// TIA Portal V18 export
FUNCTION_BLOCK "P01_TCP_Com"   // FB12, LAD
{ S7_Optimized_Access := 'FALSE' }
// stored: SetENOAutomatically false
   VAR_INPUT
      I_Modbus_Slave_Addr : Byte;
      I_Start : Bool;
      I_Frequency : Real;   // 0-100（%）
   END_VAR
   VAR
      FB_Always_True : Bool;
      Start_TSEND_C { S7_SetPoint := 'True'} : TSEND_C;
      Frequency_TSNED_C { S7_SetPoint := 'True'} : TSEND_C;
      P1 : Bool;
      P2 : Bool;
      Start_T { S7_SetPoint := 'True'} : TON_TIME;
      Stop_T { S7_SetPoint := 'True'} : TOF_TIME;
      Command_Start { S7_SetPoint := 'True'} : Bool;
      Command_Stop { S7_SetPoint := 'True'} : Bool;
      Command_Freq { S7_SetPoint := 'True'} : Bool;
      Start_Array : Array[0..5] of Byte;
      Stop_Array : Array[0..5] of Byte;
      Freq_Array : Array[0..8] of Byte;
      CRC_Result : Word;
      "TSEND_DATA_Start/Stop" : Array[0..7] of Byte;
      TSEND_DATA_Freq : Array[0..10] of Byte;
      Start_TSEND_Rescan_T { S7_SetPoint := 'True'} : TON_TIME;
      Frequency_TSEND_Rescan_T { S7_SetPoint := 'True'} : TON_TIME;
      LGF_Impulse_Instance { S7_SetPoint := 'True'} : "LGF_Impulse";
   END_VAR
   VAR_TEMP
      T_Start_TSEND : Bool;
      T_Stop_TSEND : Bool;
      T_Frequency_TSEND : Bool;
      T_Frequency : Word;
   END_VAR
   // Start_Array[0] := 16#01;
   // Start_Array[1] := 16#05;
   // Start_Array[2] := 16#00;
   // Start_Array[3] := 16#04;
   // Start_Array[4] := 16#FF;
   // Start_Array[5] := 16#00;
   // Stop_Array[0] := 16#01;
   // Stop_Array[1] := 16#05;
   // Stop_Array[2] := 16#00;
   // Stop_Array[3] := 16#04;
   // Stop_Array[4..5] := 16#00;
   // Freq_Array[0] := 16#01;
   // Freq_Array[1] := 16#10;
   // Freq_Array[2] := 16#00;
   // Freq_Array[3] := 16#08;
   // Freq_Array[4] := 16#00;
   // Freq_Array[5] := 16#01;
   // Freq_Array[6] := 16#02;
   // Freq_Array[7] := 16#00;
   // Freq_Array[8] := 16#64;
   VAR_TEMP   // added for the SCL form of the ladder/FBD networks
      _w1 : Bool;
      _w2 : Bool;
      _w3 : Bool;
   END_VAR
BEGIN

REGION Network 1: FBAT
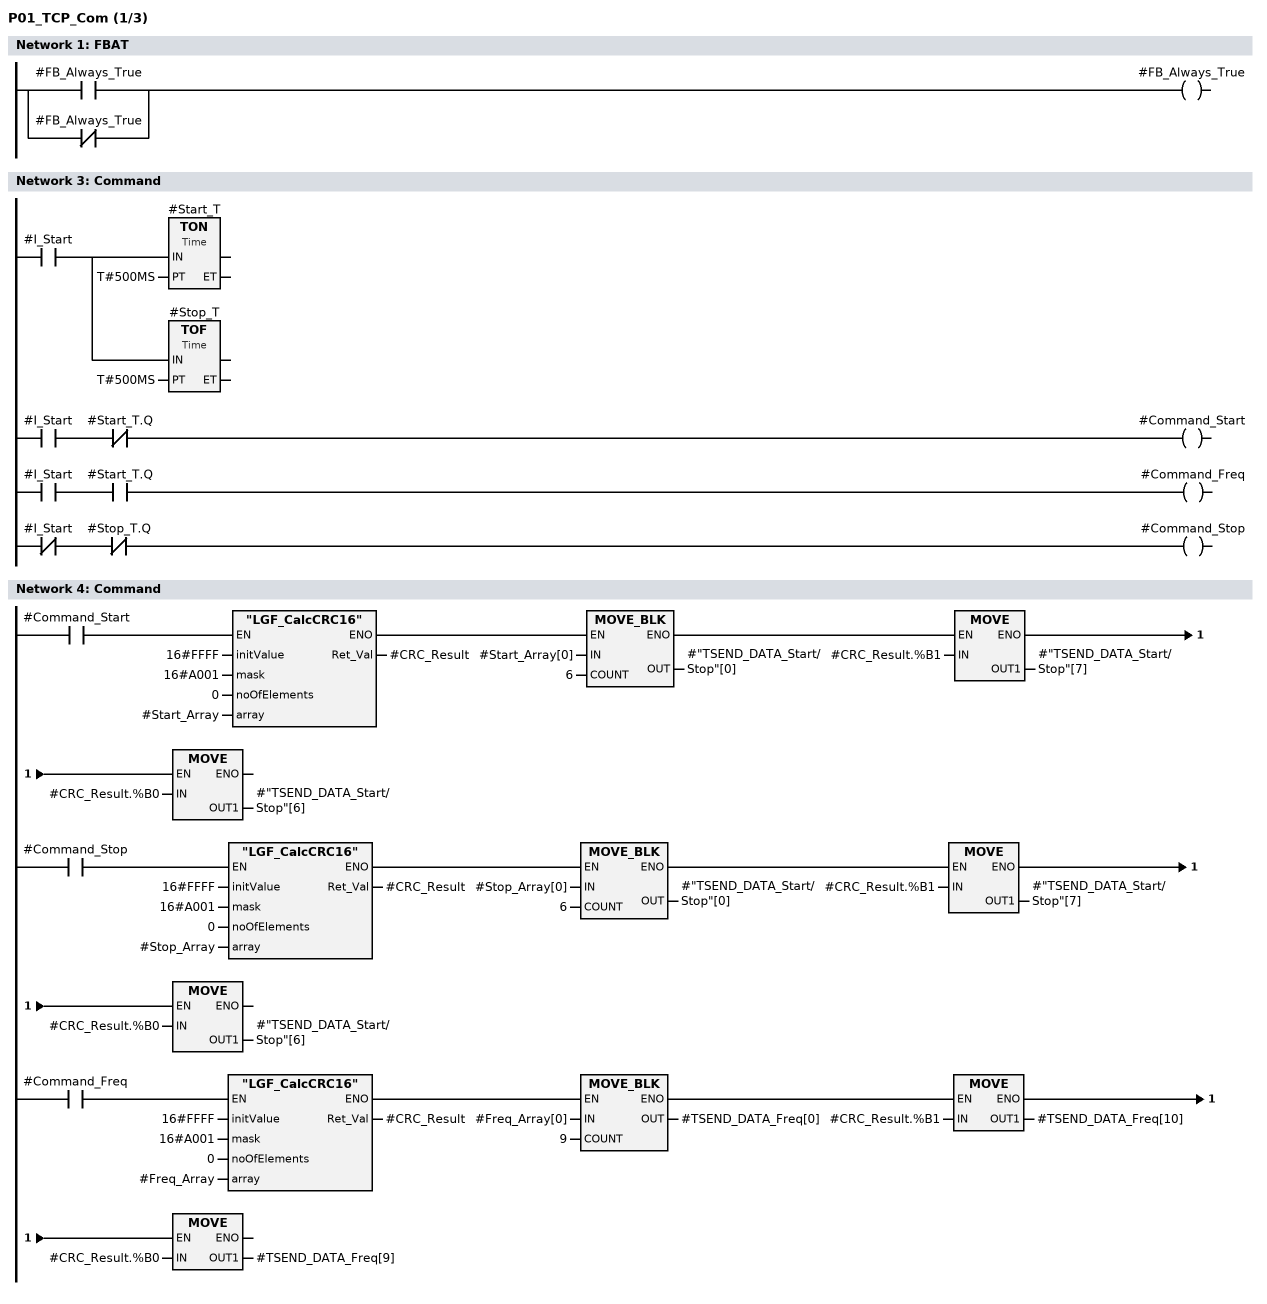
   RUNG wire#powerrail
      Contact( #FB_Always_True )
      wire#w1
      Coil( #FB_Always_True )
   END_RUNG
   RUNG wire#powerrail
      I_Contact( #FB_Always_True )
   END_RUNG wire#w1
   // the same network as SCL:
   #FB_Always_True := #FB_Always_True OR NOT #FB_Always_True;
END_REGION

REGION Network 2 (SCL): Parameter Transform
   #T_Frequency := ROUND(#I_Frequency * 5.0); //Frequency Transform
   #Freq_Array[7] := #T_Frequency.%B1;
   #Freq_Array[8] := #T_Frequency.%B0;
END_REGION

REGION Network 3: Command
   RUNG wire#powerrail
      Contact( #I_Start )
      wire#w1
      { S7_Templates := "time_type := Time" } #Start_T.TON(pt := T#500MS, et =>)
   END_RUNG
   RUNG wire#w1
      { S7_Templates := "time_type := Time" } #Stop_T.TOF(pt := T#500MS, et =>)
   END_RUNG
   RUNG wire#powerrail
      Contact( #I_Start )
      I_Contact( #Start_T.Q )
      Coil( #Command_Start )
   END_RUNG
   RUNG wire#powerrail
      Contact( #I_Start )
      Contact( #Start_T.Q )
      Coil( #Command_Freq )
   END_RUNG
   RUNG wire#powerrail
      I_Contact( #I_Start )
      I_Contact( #Stop_T.Q )
      Coil( #Command_Stop )
   END_RUNG
   // the same network as SCL:
   #Start_T(IN := #I_Start, PT := T#500MS);   // TON
   #Stop_T(IN := #I_Start, PT := T#500MS);   // TOF
   #Command_Start := #I_Start AND NOT #Start_T.Q;
   #Command_Freq := #I_Start AND #Start_T.Q;
   #Command_Stop := NOT #I_Start AND NOT #Stop_T.Q;
END_REGION

REGION Network 4: Command
   #CRC_Result := "LGF_CalcCRC16"(EN := #Command_Start,
                           initValue := 16#FFFF,
                           mask := 16#A001,
                           noOfElements := 0,
                           "array" := #Start_Array,
                           ENO => #_w1);
   IF #_w1 THEN
       MOVE_BLK(IN := #Start_Array[0], COUNT := 6, OUT => #"TSEND_DATA_Start/Stop"[0]);
       #"TSEND_DATA_Start/Stop"[7] := #CRC_Result.%B1;
       #"TSEND_DATA_Start/Stop"[6] := #CRC_Result.%B0;
   END_IF;
   #CRC_Result := "LGF_CalcCRC16"(EN := #Command_Stop,
                           initValue := 16#FFFF,
                           mask := 16#A001,
                           noOfElements := 0,
                           "array" := #Stop_Array,
                           ENO => #_w2);
   IF #_w2 THEN
       MOVE_BLK(IN := #Stop_Array[0], COUNT := 6, OUT => #"TSEND_DATA_Start/Stop"[0]);
       #"TSEND_DATA_Start/Stop"[7] := #CRC_Result.%B1;
       #"TSEND_DATA_Start/Stop"[6] := #CRC_Result.%B0;
   END_IF;
   #CRC_Result := "LGF_CalcCRC16"(EN := #Command_Freq,
                           initValue := 16#FFFF,
                           mask := 16#A001,
                           noOfElements := 0,
                           "array" := #Freq_Array,
                           ENO => #_w3);
   IF #_w3 THEN
       MOVE_BLK(IN := #Freq_Array[0], COUNT := 9, OUT => #TSEND_DATA_Freq[0]);
       #TSEND_DATA_Freq[10] := #CRC_Result.%B1;
       #TSEND_DATA_Freq[9] := #CRC_Result.%B0;
   END_IF;
END_REGION

REGION Network 5
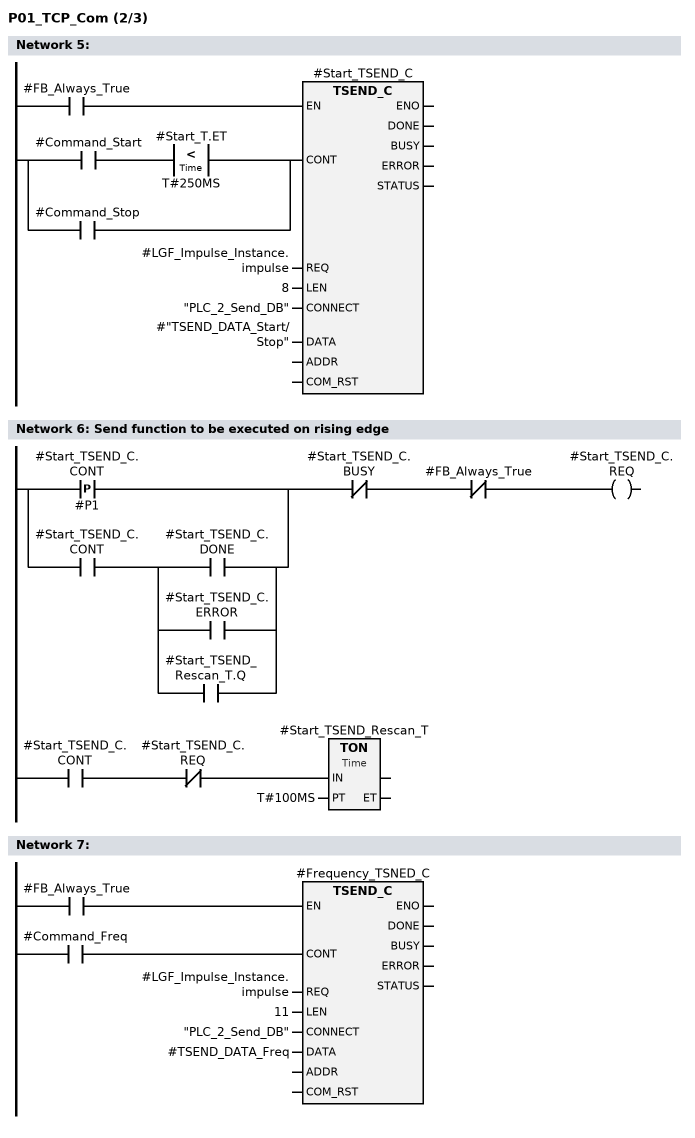
   RUNG wire#powerrail
      Contact( #FB_Always_True )
      #Start_TSEND_C.TSEND_C(CONT := wire#w1, REQ := #LGF_Impulse_Instance.impulse, LEN := 8, CONNECT := "PLC_2_Send_DB", DATA := #"TSEND_DATA_Start/Stop", ADDR :=, COM_RST :=, DONE =>, BUSY =>, ERROR =>, STATUS =>)
   END_RUNG
   RUNG wire#powerrail
      Contact( #Command_Start )
      { S7_Templates := "SrcType := Time" } LT_Contact(in1 := #Start_T.ET, in2 := T#250MS)
   END_RUNG wire#w1
   RUNG wire#powerrail
      Contact( #Command_Stop )
   END_RUNG wire#w1
   // the same network as SCL:
   IF #FB_Always_True THEN
       #Start_TSEND_C(CONT := (#Command_Start AND (#Start_T.ET < T#250MS)) OR #Command_Stop,   // TSEND_C
                      REQ := #LGF_Impulse_Instance.impulse,
                      LEN := 8,
                      CONNECT := "PLC_2_Send_DB",
                      DATA := #"TSEND_DATA_Start/Stop");
   END_IF;
END_REGION

REGION Network 6: Send function to be executed on rising edge
   RUNG wire#powerrail
      P_Contact(operand := #Start_TSEND_C.CONT, bit := #P1)
      wire#w1
      I_Contact( #Start_TSEND_C.BUSY )
      I_Contact( #FB_Always_True )
      Coil( #Start_TSEND_C.REQ )
   END_RUNG
   RUNG wire#powerrail
      Contact( #Start_TSEND_C.CONT )
      wire#w2
      Contact( #Start_TSEND_C.DONE )
   END_RUNG wire#w1
   RUNG wire#w2
      Contact( #Start_TSEND_C.ERROR )
   END_RUNG wire#w1
   RUNG wire#w2
      Contact( #Start_TSEND_Rescan_T.Q )
   END_RUNG wire#w1
   RUNG wire#powerrail
      Contact( #Start_TSEND_C.CONT )
      I_Contact( #Start_TSEND_C.REQ )
      { S7_Templates := "time_type := Time" } #Start_TSEND_Rescan_T.TON(pt := T#100MS, et =>)
   END_RUNG
   // the same network as SCL:
   #_w1 := #Start_TSEND_C.CONT AND NOT #P1;   // rising edge of #Start_TSEND_C.CONT
   #P1 := #Start_TSEND_C.CONT;
   #Start_TSEND_C.REQ := (#_w1 OR (#Start_TSEND_C.CONT AND (#Start_TSEND_C.DONE OR #Start_TSEND_C.ERROR OR #Start_TSEND_Rescan_T.Q))) AND NOT #Start_TSEND_C.BUSY AND NOT #FB_Always_True;
   #Start_TSEND_Rescan_T(IN := #Start_TSEND_C.CONT AND NOT #Start_TSEND_C.REQ, PT := T#100MS);   // TON
END_REGION

REGION Network 7
   RUNG wire#powerrail
      Contact( #FB_Always_True )
      #Frequency_TSNED_C.TSEND_C(CONT := wire#w1, REQ := #LGF_Impulse_Instance.impulse, LEN := 11, CONNECT := "PLC_2_Send_DB", DATA := #TSEND_DATA_Freq, ADDR :=, COM_RST :=, DONE =>, BUSY =>, ERROR =>, STATUS =>)
   END_RUNG
   RUNG wire#powerrail
      Contact( #Command_Freq )
   END_RUNG wire#w1
   // the same network as SCL:
   IF #FB_Always_True THEN
       #Frequency_TSNED_C(CONT := #Command_Freq,   // TSEND_C
                          REQ := #LGF_Impulse_Instance.impulse,
                          LEN := 11,
                          CONNECT := "PLC_2_Send_DB",
                          DATA := #TSEND_DATA_Freq);
   END_IF;
END_REGION

REGION Network 8: Send function to be executed on rising edge
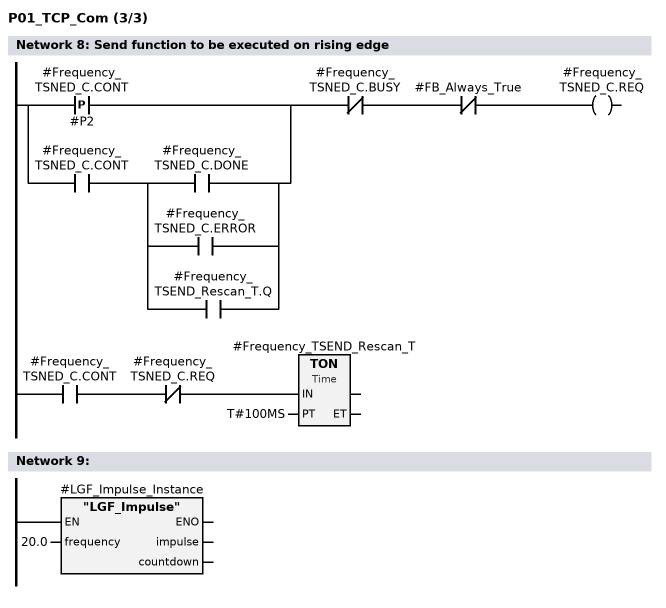
   RUNG wire#powerrail
      P_Contact(operand := #Frequency_TSNED_C.CONT, bit := #P2)
      wire#w1
      I_Contact( #Frequency_TSNED_C.BUSY )
      I_Contact( #FB_Always_True )
      Coil( #Frequency_TSNED_C.REQ )
   END_RUNG
   RUNG wire#powerrail
      Contact( #Frequency_TSNED_C.CONT )
      wire#w2
      Contact( #Frequency_TSNED_C.DONE )
   END_RUNG wire#w1
   RUNG wire#w2
      Contact( #Frequency_TSNED_C.ERROR )
   END_RUNG wire#w1
   RUNG wire#w2
      Contact( #Frequency_TSEND_Rescan_T.Q )
   END_RUNG wire#w1
   RUNG wire#powerrail
      Contact( #Frequency_TSNED_C.CONT )
      I_Contact( #Frequency_TSNED_C.REQ )
      { S7_Templates := "time_type := Time" } #Frequency_TSEND_Rescan_T.TON(pt := T#100MS, et =>)
   END_RUNG
   // the same network as SCL:
   #_w1 := #Frequency_TSNED_C.CONT AND NOT #P2;   // rising edge of #Frequency_TSNED_C.CONT
   #P2 := #Frequency_TSNED_C.CONT;
   #Frequency_TSNED_C.REQ := (#_w1 OR (#Frequency_TSNED_C.CONT AND (#Frequency_TSNED_C.DONE OR #Frequency_TSNED_C.ERROR OR #Frequency_TSEND_Rescan_T.Q))) AND NOT #Frequency_TSNED_C.BUSY AND NOT #FB_Always_True;
   #Frequency_TSEND_Rescan_T(IN := #Frequency_TSNED_C.CONT AND NOT #Frequency_TSNED_C.REQ, PT := T#100MS);   // TON
END_REGION

REGION Network 9
   RUNG wire#powerrail
      #LGF_Impulse_Instance(frequency := 20.0, impulse =>, countdown =>)
   END_RUNG
   // the same network as SCL:
   #LGF_Impulse_Instance(frequency := 20.0);   // "LGF_Impulse"
END_REGION
END_FUNCTION_BLOCK
